(*
	Check if all test suites are finished.
*)
FUNCTION IS_ALL_FINISHED : BOOL

IS_ALL_FINISHED :=		GVL_TcUnit.TcUnitRunner.AllTestSuitesFinished
					AND GVL_TcUnit.TcUnitRunner.TestResults.StoredGeneralTestResults;

END_FUNCTION

(* stored: Version 1.1.0.1, ProductVersion 3.1.4024.11
   POU IS_ALL_FINISHED: Id {9ca4f606-3466-47c8-b88b-dc63180080b3}, SpecialFunc None *)
